FUNCTION_BLOCK MotionEnable
VAR_INPUT
END_VAR
VAR_OUTPUT
END_VAR
VAR
END_VAR

END_FUNCTION_BLOCK

(* stored: Version 1.1.0.1, ProductVersion 3.1.4024.4
   POU MotionEnable: Id {168e200a-6624-4037-8d35-a43cb7583681}, SpecialFunc None *)
